# EPICS IOC start-up script: soft_iocs/srs/iocBoot/iocsr570/SR_570.iocsh
# ### SR_570.iocsh ###

#- ###################################################
#- PREFIX         - IOC Prefix
#- INSTANCE       - Instance Prefix
#- PORT           - Serial port name
#- IP             - Location of IP module
#- ###################################################

#- Stanford Research Systems SR570 Current Preamplifier
asynOctetSetInputEos( "$(PORT)", -1, "\r")
asynOctetSetOutputEos("$(PORT)", -1, "\r")

dbLoadRecords("$(IP)/ipApp/Db/SR570.db", "P=$(PREFIX),A=$(INSTANCE),PORT=$(PORT)")
